# B&R Automation Studio project X20CP1382
Automation Studio 4.12.3.127 SP; technology packages: mappView 5.24.4

## Configuration Config1

CPU X20CP1382, AutomationRuntime D4.83, Build 4.1.2, Vc V4.72.3

## Logical view

### Program Logical/Program

#### Variables.var
```iecst
(*Automatik*)
VAR
	rAsiStart : r_trig;
	rChangeMode : r_trig;
	bAutoMode : BOOL;
	bAutomodeChange : BOOL;
	bGondelsNotEmpty : BOOL;
	bLightGreen : BOOL;
	bLightRed : BOOL;
	bManualFast : BOOL;
	RisingLightBarrier : r_trig;
END_VAR
(*Handbetrieb*)
VAR
	bManualMode : BOOL;
	bManualNormal : BOOL;
	bManualSlow : BOOL;
	bManualStart : BOOL;
	bManualStop : BOOL;
	bModuloBusy : BOOL;
	bNextRFID : BOOL;
	bNotSetup : BOOL;
	bResetPersonInGondel : BOOL;
	bSafetyResetReq : {REDUND_UNREPLICABLE} BOOL;
	bSetAllGondels : BOOL := FALSE;
	bSetup : {REDUND_UNREPLICABLE} BOOL;
	bSkipAutoChange : BOOL;
	bStartModulo : BOOL;
	bVisuPushBetrieb : BOOL;
END_VAR
(*Lichter*)
VAR
	tonQuit : TON; (*Blinken Licht Start Asi*)
	tonStart : TON; (*Blinken Licht Quit Asi*)
	bVisuSpotLeft : BOOL;
	bVisuSpotRight : BOOL;
	eAutoControl : E_AutoControl;
	eSpeed : E_Speed := 0;
	i : INT; (*Schleifenvariable*)
	nLastRFID : UINT;
	nColor : USINT;
	tonManualSwitch : TON;
	nCurrentPerson : INT;
	nGondelValueSet : USINT;
	nLastRFIDAuto : UINT;
	nLEDVisu : INT;
END_VAR
(*RFID/ Gondels*)
VAR
	aPersonInCarIs : ARRAY[0..5] OF USINT;
	aPersonInCarSet : ARRAY[0..5] OF USINT;
	aRFIDColors : ARRAY[0..5] OF INT;
	aVisuRFIDCol : ARRAY[0..5] OF BOOL;
	nRFIDArrIndex : USINT;
	nSpinnCountIs : USINT;
	nSpinnCountSet : USINT;
END_VAR
(*Safety*)
VAR
	rfAutomode : RF_TRIG;
	rAsiQuit : r_trig;
	rSetup : {REDUND_UNREPLICABLE} r_trig;
	rRFIDTrack : r_trig;
END_VAR
(*Visualisierung*)
VAR
	rTrigGreen : r_trig;
	rTrigModulo : r_trig;
	rTrigRed : r_trig;
	sDisplayVisu : {REDUND_UNREPLICABLE} STRING[80];
	sManualColor : STRING[80];
	sVisuDrehrichtung : STRING[80];
	sVisuMode : STRING[80];
	tonTimerRun : TON;
END_VAR
```

#### Cyclic.st
```iecst
PROGRAM _CYCLIC
	Safety;

	rChangeMode.CLK:=gButtonOnOff OR bManualStart;
	IF rChangeMode.Q AND NOT bSafetyResetReq THEN
		bAutoMode := NOT bAutoMode;
	END_IF

	IF bGondelsNotEmpty THEN
		bAutoMode:=FALSE;
	END_IF

	IF bSetup AND NOT bSafetyResetReq AND bAutoMode THEN
		Setup;
	ELSIF bAutoMode AND NOT bSetup AND NOT bSafetyResetReq THEN
		Automatic;
	END_IF

	IF NOT bAutoMode AND NOT bSafetyResetReq THEN
		Manual;
	END_IF

	Drive;
	Display;
	Lights;
	Visu;
	rChangeMode();
	bNotSetup:= NOT bSetup;
	bManualMode:=NOT bAutoMode;

END_PROGRAM
```

#### Lights.st
```iecst
ACTION Lights:

	gLED1:=0;
	gLED2:=0;
	gLED3:=0;
	gLED4:=0;

	CASE nLEDVisu OF
		1:
			gLED1:=TRUE;
		2:
			gLED2:=TRUE;
		3:
			gLED1:=TRUE;
			gLED2:=TRUE;
		4:
			gLED3:=TRUE;
		5:
			gLED1:=TRUE;
			gLED3:=TRUE;
		6:
			gLED2:=TRUE;
			gLED3:=TRUE;
		7:
			gLED1:=TRUE;
			gLED2:=TRUE;
			gLED3:=TRUE;
		8:
			gLED4:=TRUE;
		9:
			gLED1:=TRUE;
			gLED4:=TRUE;
		10:
			gLED2:=TRUE;
			gLED4:=TRUE;
		11:
			gLED1:=TRUE;
			gLED2:=TRUE;
			gLED4:=TRUE;
		12:
			gLED3:=TRUE;
			gLED4:=TRUE;
		13:
			gLED1:=TRUE;
			gLED3:=TRUE;
			gLED4:=TRUE;
		14:
			gLED2:=TRUE;
			gLED3:=TRUE;
			gLED4:=TRUE;
		15:
			gLED1:=TRUE;
			gLED2:=TRUE;
			gLED3:=TRUE;
			gLED4:=TRUE;
		END_CASE

	IF bVisuSpotLeft THEN
		gSpotlightLeft:=TRUE;
	ELSE
		gSpotlightLeft:=FALSE;
	END_IF

	IF bVisuSpotRight THEN
		gSpotlightRight:=TRUE;
	ELSE
		gSpotlightRight:=FALSE;
	END_IF

END_ACTION
```

#### Manual.st
```iecst
ACTION Manual:
	gASILight1:=FALSE;

	IF bVisuPushBetrieb THEN
		eSpeed:=stop;
	END_IF
		IF gButtonStop OR bManualStop THEN
			eSpeed:=stop;
		ELSIF (gButtonSlow AND gButtonFast) OR bManualNormal THEN
			eSpeed:=normal;
		ELSIF gButtonFast OR bManualFast THEN
			eSpeed:=fast;
		ELSIF gButtonSlow OR bManualSlow THEN
			eSpeed:=slow;
		END_IF

	IF sManualColor = '0' THEN
		nColor:=0;
	ELSIF sManualColor = '1' THEN
		nColor:=1;
	ELSIF sManualColor='2' THEN
		nColor:=2;
	ELSIF sManualColor='3' THEN
		nColor:=3;
	ELSIF sManualColor='4' THEN
		nColor:=4;
	ELSIF sManualColor='5' THEN
		nColor:=5;
	END_IF
	rTrigModulo.CLK:=bStartModulo;
	IF rTrigModulo.Q THEN
		eSpeed:=slow;
		bModuloBusy:=TRUE;
	END_IF
	IF bModuloBusy AND gRFIDColor = aRFIDColors[nColor] THEN
		eSpeed:=stop;
		bModuloBusy:=FALSE;

	END_IF

	tonManualSwitch.IN:=gButtonStop;
	tonManualSwitch.PT:=T#5s;
	IF tonManualSwitch.Q THEN
		gDriveDirection:=NOT gDriveDirection;
		tonManualSwitch.IN:=FALSE;
	END_IF

	IF bResetPersonInGondel THEN
		aPersonInCarIs[nRFIDArrIndex]:=0;
	END_IF
	IF eSpeed <> stop THEN
		gLightGreen:=FALSE;
		gLightRed:=TRUE;
	ELSIF rTrigGreen.Q THEN
		gLightGreen:=NOT gLightGreen;
	ELSIF rTrigRed.Q THEN
		gLightRed:= NOT gLightRed;
	END_IF

	IF aPersonInCarIs[0]<> 0 OR aPersonInCarIs[1]<> 0 OR aPersonInCarIs[2]<> 0 OR aPersonInCarIs[3]<> 0 OR aPersonInCarIs[4]<> 0 OR aPersonInCarIs[5]<> 0 OR aPersonInCarIs[0]<> 0 THEN
		bGondelsNotEmpty:=TRUE;
	ELSE
			bGondelsNotEmpty:=FALSE;
	END_IF

	tonManualSwitch();
	rTrigModulo();
	rTrigGreen(CLK:=bLightGreen);
	rTrigRed(CLK:=bLightRed);
END_ACTION
```

#### Safety.st
```iecst
ACTION Safety:
	gEmergencyStop:= (NOT gEmergencyStop1 AND NOT gEmergencyStop2 AND NOT gEmergencyStop3 AND NOT gEmergencyStop4);

	gLightGrid:=  (NOT gLightGrid1 AND NOT gLightGrid2 AND NOT gLightGrid3 AND NOT gLightGrid4);

	gSafetyStop:=gEmergencyStop OR gLightGrid;

	//Togglen der Lampe einfügen für bessere Sichtbarkeit
	IF gSafetyStop THEN
		bSafetyResetReq := TRUE;
		eSpeed:=stop;
	END_IF

	IF rfAutomode.Q AND NOT bSkipAutoChange THEN
		bSafetyResetReq:=TRUE;
		bAutomodeChange:=TRUE;
		gASILight1:=FALSE;
		eSpeed:=stop;
	ELSIF rChangeMode.Q AND bSkipAutoChange THEN
		bSkipAutoChange:=FALSE;
		eSpeed:=stop;
	END_IF

	IF bSafetyResetReq AND tonQuit.Q THEN
		gASILight3:=NOT gASILight3;
		gASILight1:=FALSE;
	END_IF

	IF rAsiQuit.Q AND NOT bAutomodeChange THEN
		bSafetyResetReq:=FALSE;
		bSetup:=TRUE;
		gASILight3:=FALSE;

		IF bAutoMode THEN
			bAutoMode:=FALSE;
			bSkipAutoChange:=TRUE;
		ELSE
			bSkipAutoChange:=FALSE;
		END_IF
	ELSIF rAsiQuit.Q AND bAutomodeChange THEN
		bSafetyResetReq:=FALSE;
		bSetup:=TRUE;
		gASILight3:=FALSE;
		bAutomodeChange:=FALSE;
	END_IF

	IF gSafetyStop OR bSafetyResetReq THEN
		gRedTop:=TRUE;
		gRedDown:=TRUE;
		gGreenDown:=FALSE;
		gGreenTop:=FALSE;
	ELSE
		gRedTop:=FALSE;
		gRedDown:=FALSE;
		gGreenDown:=TRUE;
		gGreenTop:=TRUE;
	END_IF
	tonQuit(IN:=(NOT tonQuit.Q), PT:=T#1s);
	rfAutomode(CLK:=bAutoMode);
	rAsiQuit(CLK:=gASIQuit);
END_ACTION
```
